Staubli VAL3: sad_project_cal.dtx

public mdesc cnst_vel = {tmax=100, rmax=100, leave=0.1, reach=0.1, blend=cartesian}
public frame fReference = {x=1365.054, y=-125.975, z=-500, fatherId=world[0]}
public jointRx Jnt_cnfg = {j3=90, j5=90, j6=90}
public tool tTool = {z=200, fatherId=flange[0], ioLink=valve1}
public pointRx Pnt_1st_lyr = {rx=-180, rz=-90, shoulder=lefty, elbow=epositive, wrist=wpositive, fatherId=fReference[0]}
